FUNCTION_BLOCK ABSTRACT RunningProgramState EXTENDS ProgramState

{attribute 'monitoring' := 'call'}
{attribute 'OPC.UA.DA.Property' := '1'}
{attribute 'OPC.UA.DA.Access' := '1'}
PROPERTY FINAL Name : STRING
GET
Name := 'Running';
END_GET
END_PROPERTY

END_FUNCTION_BLOCK

(* stored: Version 1.1.0.1
   POU RunningProgramState: Id {9c9f25b8-88d5-4d9f-95d2-e187fffc78c8}, SpecialFunc None
   Property Name: Id {62c20930-e33d-49fe-970d-a9da268660ee}
   Get Get: Id {248a9be7-cc06-458d-b07d-65abc8d73e3b} *)
